# B&R Automation Studio project elevator
Automation Studio 4.2.1.214; Default project

## Configuration Simulation

CPU , AutomationRuntime D4.21

### Hardware
```
PC_any : PC_any v1.1.0.0 (OrderNumber=PC)
  Connector IF3:
    Vnc1
    VncVcObjectName1 = demo
    VncKeyMappingFile1 = VC\PS2-Keyboard.dis
  Cyclic1Duration = 100000
  Cyclic1Tolerance = 10000000
  Cyclic2Duration = 200000
  Cyclic2Tolerance = 10000000
  Cyclic3Duration = 500000
  Cyclic3Tolerance = 10000000
  Cyclic4Duration = 1000000
  Cyclic4Tolerance = 10000000
  Cyclic5Duration = 2000000
  Cyclic5Tolerance = 10000000
  Cyclic6Duration = 3000000
  Cyclic6Tolerance = 12000000
  Cyclic7Duration = 4000000
  Cyclic7Tolerance = 12000000
  Cyclic8Duration = 5000000
  Cyclic8Tolerance = 30000000
```

## Logical view

Binary libraries used (declarations not repeated): Runtime, Operator, AsIecCon, astime, standard, sys_lib, brsystem

### Global.typ - Global data types
```iecst
(*********************************************************************************
 * Copyright:
 * Author:    Chen
 * Created:   April 23, 2016/7:59 PM
 *********************************************************************************
 * Declaration of global data types
 *********************************************************************************)

TYPE

 (*电梯井接口信号定义*)
tTower_Interface: STRUCT

		Sensor_DoorOpened : BOOL;(*传感器信号指示轿厢门已打开*)
		Sensor_DoorClosed : BOOL;(*传感器信号指示轿厢门已关闭*)

		Sensor_Floor1Approached :  BOOL;(*传感器信号指示轿厢已到达对应楼层*)
		Sensor_Floor2Approached :  BOOL;
		Sensor_Floor3Approached :  BOOL;
		Sensor_Floor4Approached :  BOOL;
		Sensor_Floor5Approached :  BOOL;
		Sensor_Floor6Approached :  BOOL;
		Sensor_Floor7Approached :  BOOL;

		Signal_Start_DoorMotor_P : BOOL; (*控制信号，上升沿触发，使轿厢门电机正转固定的角度，打开轿厢门*)
		Signal_Start_DoorMotor_N : BOOL; (*控制信号，上升沿触发，使轿厢门电机反转固定的角度，关闭轿厢门*)

		Signal_Start_CabinMotor_P : BOOL; (*控制信号，上升沿触发，使轿厢提升电机正转，电梯上行*)
		Signal_Start_CabinMotor_N : BOOL; (*控制信号，上升沿触发，使轿厢提升电机反转，电梯下行*)
		Signal_Stop_CabinMotor : BOOL;    (*控制信号，上升沿触发，使轿厢提升电机停止*)

		Sensor_Position_Door : UINT;	  (*轿厢门位置反馈*)
		Sensor_Position_Cabin : UINT;     (*轿厢垂直位置反馈*)

END_STRUCT;

(*楼层面板接口信号定义*)
tFloor_Interface: STRUCT
		Key_Up : BOOL;(*向上按钮*)
		Key_Down : BOOL;(*向下按钮*)
		Display_Current_Floor_Left : USINT;(*左电梯当前楼层显示数码管*)
		Display_Current_Floor_Right : USINT;(*右电梯当前楼层显示数码管*)
		Display_Current_Direction_Left : STRING[2];(*左电梯当前运行方向显示数码管*)
		Display_Current_Direction_Right : STRING[2];(*右电梯当前运行方向显示数码管*)
		Display_UpSelected : tCheckStatus; (*电梯向上按钮指示灯*)
		Display_DownSelected : tCheckStatus; (*电梯向下按钮指示灯*)
END_STRUCT;

(*对应楼层的设置状态*)
tCheckStatus :
		(
		Checked:=16#3340,
		UnChecked:=16#FE10
);

(*轿厢接口信号定义*)
tCabin_Interface: STRUCT

		Key_Open : BOOL; (*开门按钮*)
		Key_Close : BOOL; (*关门按钮*)
		Key_Floor1 : BOOL; (*目标楼层按钮*)
		Key_Floor2 : BOOL;
		Key_Floor3 : BOOL;
		Key_Floor4 : BOOL;
		Key_Floor5 : BOOL;
		Key_Floor6 : BOOL;
		Key_Floor7 : BOOL;
		Display_Floor1Selected : tCheckStatus;(*目标楼层被选中指示灯*)
		Display_Floor2Selected : tCheckStatus;
		Display_Floor3Selected : tCheckStatus;
		Display_Floor4Selected : tCheckStatus;
		Display_Floor5Selected : tCheckStatus;
		Display_Floor6Selected : tCheckStatus;
		Display_Floor7Selected : tCheckStatus;

		Display_Current_Floor : USINT;  (*当前楼层显示数码管*)
		Display_Current_Direction : STRING[2];    (*当前运行方向显示数码管*)

END_STRUCT;

END_TYPE
```

### Global.var - Global variables
```iecst
(*********************************************************************************
 * Copyright:
 * Author:    Chen
 * Created:   April 23, 2016/7:59 PM
 *********************************************************************************
 * Declaration of global variables
 *********************************************************************************)
VAR
	LeftTower : tTower_Interface; (*实例化左电梯井接口*)
	RightTower : tTower_Interface; (*实例化右电梯井接口*)
	LeftCabin : tCabin_Interface; (*实例化左电梯轿厢接口*)
	RightCabin : tCabin_Interface; (*实例化右电梯轿厢接口*)
	FloorPanel : ARRAY[0..6] OF tFloor_Interface := [7(0)];
END_VAR
```


### Program Logical/Model (IEC)

#### Cyclic.st - Cyclic code
```iecst
PROGRAM _CYCLIC

	(*左电梯轿厢门状态机*)
	CASE LeftDoorState OF
		DoorIsClosed:
			IF LeftTower.Signal_Start_DoorMotor_P   THEN
				LeftTower.Sensor_DoorClosed := FALSE;
				LeftDoorState := DoorIsOpening;

			END_IF
		DoorIsOpened:
			IF LeftTower.Signal_Start_DoorMotor_N   THEN
				LeftTower.Sensor_DoorOpened := FALSE;
				LeftDoorState := DoorIsClosing;
			END_IF
		DoorIsClosing:
			IF LeftTower.Sensor_Position_Door > 0 THEN
				LeftTower.Sensor_Position_Door := LeftTower.Sensor_Position_Door-1;
			ELSE
				LeftTower.Sensor_DoorClosed := TRUE;
				LeftDoorState := DoorIsClosed;
			END_IF
		DoorIsOpening:
			IF LeftTower.Sensor_Position_Door < 50 THEN
				LeftTower.Sensor_Position_Door := LeftTower.Sensor_Position_Door+1;
			ELSE
				LeftTower.Sensor_DoorOpened := TRUE;
				LeftDoorState := DoorIsOpened;
			END_IF
	END_CASE

	(*左电梯轿厢运动状态机*)

	CASE LeftCabinState OF
		CabinIsStoped:
			IF LeftTower.Signal_Start_CabinMotor_P   THEN
				LeftCabinState := CabinIsGoingUp;
			ELSIF LeftTower.Signal_Start_CabinMotor_N THEN
				LeftCabinState := CabinIsGoingDown;
			END_IF
			LeftCabin.Display_Current_Direction := '--';
			FOR i := 0 TO 6 DO
				FloorPanel[i].Display_Current_Direction_Left := '--';
			END_FOR
		CabinIsGoingUp:
			IF LeftTower.Sensor_Position_Cabin < 600 THEN
			    LeftTower.Sensor_Position_Cabin := LeftTower.Sensor_Position_Cabin+1;
			END_IF
			IF  LeftTower.Signal_Stop_CabinMotor   THEN
				LeftCabinState := CabinIsStoped;
			END_IF
			LeftCabin.Display_Current_Direction := '/\';
			FOR i := 0 TO 6 DO
				FloorPanel[i].Display_Current_Direction_Left := '/\';
			END_FOR

		CabinIsGoingDown:
			IF LeftTower.Sensor_Position_Cabin > 0 THEN
				LeftTower.Sensor_Position_Cabin := LeftTower.Sensor_Position_Cabin-1;
			END_IF
			IF  LeftTower.Signal_Stop_CabinMotor   THEN
				LeftCabinState := CabinIsStoped;
			END_IF
			LeftCabin.Display_Current_Direction := '\/';
			FOR i := 0 TO 6 DO
				FloorPanel[i].Display_Current_Direction_Left := '\/';
			END_FOR

		END_CASE

	IF LeftTower.Sensor_Position_Cabin = 0 THEN
		LeftTower.Sensor_Floor1Approached := TRUE;
	ELSE
		LeftTower.Sensor_Floor1Approached := FALSE;
	END_IF

	IF LeftTower.Sensor_Position_Cabin = 100 THEN
		LeftTower.Sensor_Floor2Approached := TRUE;
	ELSE
		LeftTower.Sensor_Floor2Approached := FALSE;
	END_IF

	IF LeftTower.Sensor_Position_Cabin = 200 THEN
		LeftTower.Sensor_Floor3Approached := TRUE;
	ELSE
		LeftTower.Sensor_Floor3Approached := FALSE;
	END_IF

	IF LeftTower.Sensor_Position_Cabin = 300 THEN
		LeftTower.Sensor_Floor4Approached := TRUE;
	ELSE
		LeftTower.Sensor_Floor4Approached := FALSE;
	END_IF
	IF LeftTower.Sensor_Position_Cabin = 400 THEN
		LeftTower.Sensor_Floor5Approached := TRUE;
	ELSE
		LeftTower.Sensor_Floor5Approached := FALSE;
	END_IF
	IF LeftTower.Sensor_Position_Cabin = 500 THEN
		LeftTower.Sensor_Floor6Approached := TRUE;
	ELSE
		LeftTower.Sensor_Floor6Approached := FALSE;
	END_IF
	IF LeftTower.Sensor_Position_Cabin = 600 THEN
		LeftTower.Sensor_Floor7Approached := TRUE;
	ELSE
		LeftTower.Sensor_Floor7Approached := FALSE;
	END_IF

	IF LeftTower.Sensor_Position_Cabin < 100 THEN
		LeftCabin.Display_Current_Floor := 1;
	ELSIF 	LeftTower.Sensor_Position_Cabin < 200 THEN
        LeftCabin.Display_Current_Floor := 2;
	ELSIF 	LeftTower.Sensor_Position_Cabin < 300 THEN
		LeftCabin.Display_Current_Floor := 3;
	ELSIF 	LeftTower.Sensor_Position_Cabin < 400 THEN
		LeftCabin.Display_Current_Floor := 4;
	ELSIF 	LeftTower.Sensor_Position_Cabin < 500 THEN
		LeftCabin.Display_Current_Floor := 5;
	ELSIF 	LeftTower.Sensor_Position_Cabin < 600 THEN
		LeftCabin.Display_Current_Floor := 6;
	ELSE
		LeftCabin.Display_Current_Floor := 7;
	END_IF

	FOR i := 0 TO 6 DO
		FloorPanel[i].Display_Current_Floor_Left := LeftCabin.Display_Current_Floor;
	END_FOR

	(*右电梯轿厢门状态机*)
	CASE RightDoorState OF
		DoorIsClosed:
			IF RightTower.Signal_Start_DoorMotor_P   THEN
				RightTower.Sensor_DoorClosed := FALSE;
				RightDoorState := DoorIsOpening;

			END_IF
		DoorIsOpened:
			IF RightTower.Signal_Start_DoorMotor_N   THEN
				RightTower.Sensor_DoorOpened := FALSE;
				RightDoorState := DoorIsClosing;
			END_IF
		DoorIsClosing:
			IF RightTower.Sensor_Position_Door > 0 THEN
				RightTower.Sensor_Position_Door := RightTower.Sensor_Position_Door-1;
			ELSE
				RightTower.Sensor_DoorClosed := TRUE;
				RightDoorState := DoorIsClosed;
			END_IF
		DoorIsOpening:
			IF RightTower.Sensor_Position_Door < 50 THEN
				RightTower.Sensor_Position_Door := RightTower.Sensor_Position_Door+1;
			ELSE
				RightTower.Sensor_DoorOpened := TRUE;
				RightDoorState := DoorIsOpened;
			END_IF
	END_CASE

	(*右电梯轿厢运动状态机*)

	CASE RightCabinState OF
		CabinIsStoped:
			IF RightTower.Signal_Start_CabinMotor_P   THEN
				RightCabinState := CabinIsGoingUp;
			ELSIF RightTower.Signal_Start_CabinMotor_N THEN
				RightCabinState := CabinIsGoingDown;
			END_IF
			RightCabin.Display_Current_Direction := '--';
			FOR i := 0 TO 6 DO
				FloorPanel[i].Display_Current_Direction_Right := '--';
			END_FOR

		CabinIsGoingUp:
			IF RightTower.Sensor_Position_Cabin < 600 THEN
				RightTower.Sensor_Position_Cabin := RightTower.Sensor_Position_Cabin+1;
			END_IF
			IF  RightTower.Signal_Stop_CabinMotor   THEN
				RightCabinState := CabinIsStoped;
			END_IF
			RightCabin.Display_Current_Direction := '/\';
			FOR i := 0 TO 6 DO
				FloorPanel[i].Display_Current_Direction_Right := '/\';
			END_FOR

		CabinIsGoingDown:
			IF RightTower.Sensor_Position_Cabin > 0 THEN
				RightTower.Sensor_Position_Cabin := RightTower.Sensor_Position_Cabin-1;
			END_IF
			IF  RightTower.Signal_Stop_CabinMotor   THEN
				RightCabinState := CabinIsStoped;
			END_IF
			RightCabin.Display_Current_Direction := '\/';
			FOR i := 0 TO 6 DO
				FloorPanel[i].Display_Current_Direction_Right := '\/';
			END_FOR

	END_CASE

	IF RightTower.Sensor_Position_Cabin = 0 THEN
		RightTower.Sensor_Floor1Approached := TRUE;
	ELSE
		RightTower.Sensor_Floor1Approached := FALSE;
	END_IF

	IF RightTower.Sensor_Position_Cabin = 100 THEN
		RightTower.Sensor_Floor2Approached := TRUE;
	ELSE
		RightTower.Sensor_Floor2Approached := FALSE;
	END_IF

	IF RightTower.Sensor_Position_Cabin = 200 THEN
		RightTower.Sensor_Floor3Approached := TRUE;
	ELSE
		RightTower.Sensor_Floor3Approached := FALSE;
	END_IF

	IF RightTower.Sensor_Position_Cabin = 300 THEN
		RightTower.Sensor_Floor4Approached := TRUE;
	ELSE
		RightTower.Sensor_Floor4Approached := FALSE;
	END_IF
	IF RightTower.Sensor_Position_Cabin = 400 THEN
		RightTower.Sensor_Floor5Approached := TRUE;
	ELSE
		RightTower.Sensor_Floor5Approached := FALSE;
	END_IF
	IF RightTower.Sensor_Position_Cabin = 500 THEN
		RightTower.Sensor_Floor6Approached := TRUE;
	ELSE
		RightTower.Sensor_Floor6Approached := FALSE;
	END_IF
	IF RightTower.Sensor_Position_Cabin = 600 THEN
		RightTower.Sensor_Floor7Approached := TRUE;
	ELSE
		RightTower.Sensor_Floor7Approached := FALSE;
	END_IF

	IF RightTower.Sensor_Position_Cabin < 100 THEN
		RightCabin.Display_Current_Floor := 1;
	ELSIF 	RightTower.Sensor_Position_Cabin < 200 THEN
		RightCabin.Display_Current_Floor := 2;
	ELSIF 	RightTower.Sensor_Position_Cabin < 300 THEN
		RightCabin.Display_Current_Floor := 3;
	ELSIF 	RightTower.Sensor_Position_Cabin < 400 THEN
		RightCabin.Display_Current_Floor := 4;
	ELSIF 	RightTower.Sensor_Position_Cabin < 500 THEN
		RightCabin.Display_Current_Floor := 5;
	ELSIF 	RightTower.Sensor_Position_Cabin < 600 THEN
		RightCabin.Display_Current_Floor := 6;
	ELSE
		RightCabin.Display_Current_Floor := 7;
	END_IF
	FOR i := 0 TO 6 DO
		FloorPanel[i].Display_Current_Floor_Right := RightCabin.Display_Current_Floor;
	END_FOR

END_PROGRAM
```

#### Init.st - Init code
```iecst
PROGRAM _INIT
	(* Insert code here *)
	LeftDoorState := DoorIsClosed;
	LeftCabinState := CabinIsStoped;

	LeftTower.Sensor_DoorClosed := TRUE;
	LeftTower.Sensor_DoorOpened := FALSE;
	LeftTower.Sensor_Floor1Approached := TRUE;
	LeftTower.Sensor_Floor2Approached := FALSE;
	LeftTower.Sensor_Floor3Approached := FALSE;
	LeftTower.Sensor_Floor4Approached := FALSE;
	LeftTower.Sensor_Floor5Approached := FALSE;
	LeftTower.Sensor_Floor6Approached := FALSE;
	LeftTower.Sensor_Floor7Approached := FALSE;
	LeftTower.Sensor_Position_Door := 0;
	LeftTower.Sensor_Position_Cabin := 0;

	LeftCabin.Display_Current_Direction := '--';
	RightCabin.Display_Current_Direction := '--';

END_PROGRAM
```

#### Types.typ - Local data types
```iecst
TYPE
tDoorState :
(
	DoorIsClosed,
	DoorIsOpened,
	DoorIsClosing,
	DoorIsOpening
);

tCabinState :
(
	CabinIsStoped,
	CabinIsGoingUp,
	CabinIsGoingDown
);
END_TYPE
```

#### Variables.var - Local variables
```iecst
VAR
	Current_Direction_Left : USINT := 1;
	Current_Direction_Right : USINT := 1;
	Current_Floor_Left : USINT := 1;
	Current_Floor_Right : USINT := 1;
	disp_direction : STRING[2] := '';
	i : USINT := 0;
	Key_Close_Left : BOOL := FALSE;
	Key_Close_Right : BOOL := FALSE;
	Key_Down_Floor1 : BOOL := FALSE;
	Key_Down_Floor2 : BOOL := FALSE;
	Key_Down_Floor3 : BOOL := FALSE;
	Key_Down_Floor4 : BOOL := FALSE;
	Key_Down_Floor5 : BOOL := FALSE;
	Key_Down_Floor6 : BOOL := FALSE;
	Key_Down_Floor7 : BOOL := FALSE;
	Key_Floor1_Left : BOOL := FALSE;
	Key_Floor1_Right : BOOL := FALSE;
	Key_Floor2_Left : BOOL := FALSE;
	Key_Floor2_Right : BOOL := FALSE;
	Key_Floor3_Left : BOOL := FALSE;
	Key_Floor3_Right : BOOL := FALSE;
	Key_Floor4_Left : BOOL := FALSE;
	Key_Floor4_Right : BOOL := FALSE;
	Key_Floor5_Left : BOOL := FALSE;
	Key_Floor5_Right : BOOL := FALSE;
	Key_Floor6_Left : BOOL := FALSE;
	Key_Floor6_Right : BOOL := FALSE;
	Key_Floor7_Left : BOOL := FALSE;
	Key_Floor7_Right : BOOL := FALSE;
	Key_Open_Left : BOOL := FALSE;
	Key_Open_Right : BOOL := FALSE;
	Key_Up_Floor1 : BOOL := FALSE;
	Key_Up_Floor2 : BOOL := FALSE;
	Key_Up_Floor3 : BOOL := FALSE;
	Key_Up_Floor4 : BOOL := FALSE;
	Key_Up_Floor5 : BOOL := FALSE;
	Key_Up_Floor6 : BOOL := FALSE;
	Key_Up_Floor7 : BOOL := FALSE;
	LeftCabinState : tCabinState;
	LeftDoorState : tDoorState;
	Position_Cabin_Left : UINT := 0;
	Position_Cabin_Right : UINT := 0;
	Position_Door_Left : UINT := 0;
	Position_Door_Right : UINT := 0;
	RightCabinState : tCabinState;
	RightDoorState : tDoorState;
	Sensor_Closed_Left : BOOL := FALSE;
	Sensor_Closed_Right : BOOL := FALSE;
	Sensor_Floor1_Left : BOOL := FALSE;
	Sensor_Floor1_Right : BOOL := FALSE;
	Sensor_Floor2_Left : BOOL := FALSE;
	Sensor_Floor2_Right : BOOL := FALSE;
	Sensor_Floor3_Left : BOOL := FALSE;
	Sensor_Floor3_Right : BOOL := FALSE;
	Sensor_Floor4_Left : BOOL := FALSE;
	Sensor_Floor4_Right : BOOL := FALSE;
	Sensor_Floor5_Left : BOOL := FALSE;
	Sensor_Floor5_Right : BOOL := FALSE;
	Sensor_Floor6_Left : BOOL := FALSE;
	Sensor_Floor6_Right : BOOL := FALSE;
	Sensor_Floor7_Left : BOOL := FALSE;
	Sensor_Floor7_Right : BOOL := FALSE;
	Sensor_Opened_Left : BOOL := FALSE;
	Sensor_Opened_Right : BOOL := FALSE;
	Target_Floor_Left : USINT := 1;
	Target_Floor_Right : USINT := 1;
END_VAR
```

- Visualisation Logical/demo (not shown)

### Program Logical/controller (IEC)

#### Variables.var
```iecst
VAR
	DownLast : USINT := 0;
	UpLast : USINT := 0;
	i : USINT := 0;
	j : USINT := 0;
	k : USINT := 0;
	UpList : ARRAY[0..6] OF USINT := [7(0)];
	DownList : ARRAY[0..6] OF USINT := [7(0)];
END_VAR
```

#### Cyclic.st
```iecst
PROGRAM _CYCLIC
	(* Insert code here *)
	(*下列代码只是为了测试*)

	LeftTower.Signal_Start_DoorMotor_P := LeftCabin.Key_Open ;
	LeftTower.Signal_Start_DoorMotor_N := LeftCabin.Key_Close ;

	RightTower.Signal_Start_DoorMotor_P := RightCabin.Key_Open ;
	RightTower.Signal_Start_DoorMotor_N := RightCabin.Key_Close ;

//refresh the UpList
	FOR i := 0 TO 6 DO
		IF UpList[i] = 0 THEN
			UpLast := i;
			EXIT;
		END_IF
	END_FOR

	FOR i := 0 TO 6 DO
		IF FloorPanel[i].Key_Up THEN
			FOR j := 0 TO 6 DO
				IF UpList[j] = i+1 THEN
					EXIT;
				END_IF
				IF j = 6 THEN
					UpList[UpLast] := i+1;
					UpLast := UpLast+1;
				END_IF
			END_FOR
		END_IF
	END_FOR
//refresh the DownList
	FOR i := 0 TO 6 DO
		IF DownList[i] = 0 THEN
			DownLast := i;
			EXIT;
		END_IF
	END_FOR

	FOR i := 0 TO 6 DO
		IF FloorPanel[i].Key_Down THEN
			FOR j := 0 TO 6 DO
				IF DownList[j] = i+1 THEN
					EXIT;
				END_IF
				IF j = 6 THEN
					DownList[DownLast] := i+1;
					DownLast := DownLast+1;
				END_IF
			END_FOR
		END_IF
	END_FOR
	IF UpList[0] <> 0 THEN
		IF LeftCabin.Display_Current_Floor < UpList[0] THEN
			LeftTower.Signal_Start_CabinMotor_P := TRUE;
			LeftTower.Signal_Start_CabinMotor_N := FALSE;
		END_IF
		IF LeftCabin.Display_Current_Floor > UpList[0] THEN
			LeftTower.Signal_Start_CabinMotor_N := TRUE;
			LeftTower.Signal_Start_CabinMotor_N := FALSE;
		END_IF
		IF LeftCabin.Display_Current_Floor = UpList[0] THEN
			LeftTower.Signal_Stop_CabinMotor := TRUE;
			LeftTower.Signal_Start_CabinMotor_P := FALSE;
			LeftTower.Signal_Start_CabinMotor_N := FALSE;
			LeftTower.Signal_Start_DoorMotor_P := TRUE;
			FOR i := 0 TO 6 DO
				UpList[i] := UpList[i+1] ;
				EXIT;
				END_FOR
		END_IF
	END_IF

//	LeftTower.Signal_Start_CabinMotor_P := FloorPanel[0].Key_Up ;
//	RightTower.Signal_Start_CabinMotor_P := FloorPanel[0].Key_Up ;
//
//	LeftTower.Signal_Start_CabinMotor_N := FloorPanel[6].Key_Down ;
//	RightTower.Signal_Start_CabinMotor_N := FloorPanel[6].Key_Down ;
//
//	LeftTower.Signal_Stop_CabinMotor := FloorPanel[3].Key_Up ;
//	RightTower.Signal_Stop_CabinMotor := FloorPanel[3].Key_Up ;

	IF LeftCabin.Display_Floor1Selected = UnChecked AND LeftCabin.Key_Floor1 =1 THEN
		LeftCabin.Display_Floor1Selected := Checked;
	END_IF
	IF LeftCabin.Display_Floor2Selected = UnChecked AND LeftCabin.Key_Floor2 =1 THEN
		LeftCabin.Display_Floor2Selected := Checked;
	END_IF
	IF LeftCabin.Display_Floor3Selected = UnChecked AND LeftCabin.Key_Floor3 =1 THEN
		LeftCabin.Display_Floor3Selected := Checked;
	END_IF
	IF LeftCabin.Display_Floor4Selected = UnChecked AND LeftCabin.Key_Floor4 =1 THEN
		LeftCabin.Display_Floor4Selected := Checked;
	END_IF
	IF LeftCabin.Display_Floor5Selected = UnChecked AND LeftCabin.Key_Floor5 =1 THEN
		LeftCabin.Display_Floor5Selected := Checked;
	END_IF
	IF LeftCabin.Display_Floor6Selected = UnChecked AND LeftCabin.Key_Floor6 =1 THEN
		LeftCabin.Display_Floor6Selected := Checked;
	END_IF
	IF LeftCabin.Display_Floor7Selected = UnChecked AND LeftCabin.Key_Floor7 =1 THEN
		LeftCabin.Display_Floor7Selected := Checked;
	END_IF

	IF RightCabin.Display_Floor1Selected = UnChecked AND RightCabin.Key_Floor1 =1 THEN
		RightCabin.Display_Floor1Selected := Checked;
	END_IF
	IF RightCabin.Display_Floor2Selected = UnChecked AND RightCabin.Key_Floor2 =1 THEN
		RightCabin.Display_Floor2Selected := Checked;
	END_IF
	IF RightCabin.Display_Floor3Selected = UnChecked AND RightCabin.Key_Floor3 =1 THEN
		RightCabin.Display_Floor3Selected := Checked;
	END_IF
	IF RightCabin.Display_Floor4Selected = UnChecked AND RightCabin.Key_Floor4 =1 THEN
		RightCabin.Display_Floor4Selected := Checked;
	END_IF
	IF RightCabin.Display_Floor5Selected = UnChecked AND RightCabin.Key_Floor5 =1 THEN
		RightCabin.Display_Floor5Selected := Checked;
	END_IF
	IF RightCabin.Display_Floor6Selected = UnChecked AND RightCabin.Key_Floor6 =1 THEN
		RightCabin.Display_Floor6Selected := Checked;
	END_IF
	IF RightCabin.Display_Floor7Selected = UnChecked AND RightCabin.Key_Floor7 =1 THEN
		RightCabin.Display_Floor7Selected := Checked;
	END_IF

END_PROGRAM
```

#### Cyclic1.ld
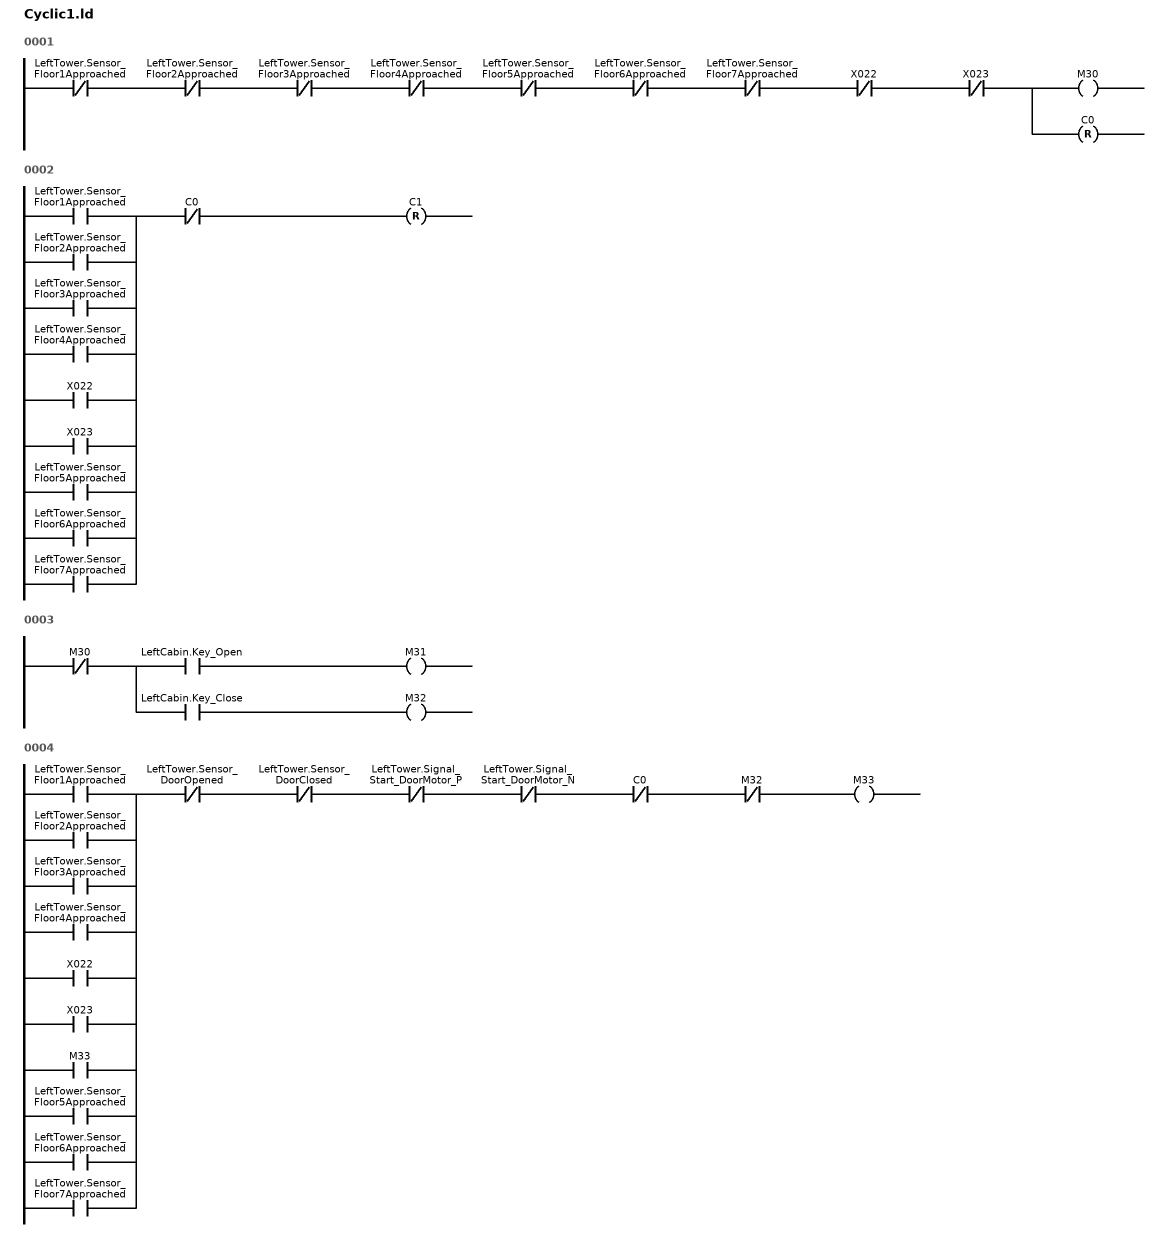
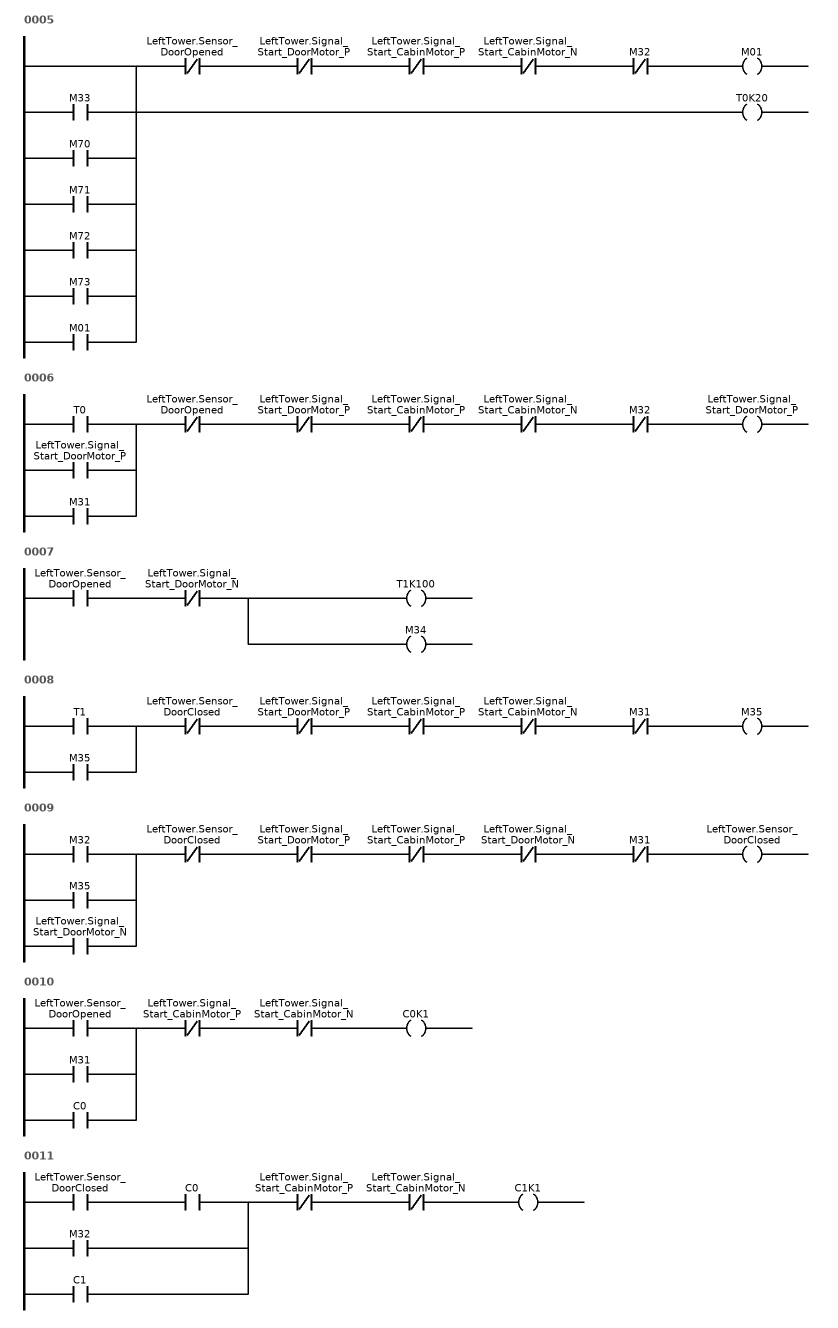
Ladder, written as Structured Text:
```iecst
PROGRAM _CYCLIC
VAR
    _p1 : BOOL;
    _z2 : BOOL;
    _z3 : BOOL;
    _z4 : BOOL;
    _z5 : BOOL;
    _z6 : BOOL;
    _z7 : BOOL;
    _p8 : BOOL;
    _p9 : BOOL;
END_VAR
(* Network 1 *)
_p1 := NOT LeftTower.Sensor_Floor1Approached AND NOT LeftTower.Sensor_Floor2Approached AND NOT LeftTower.Sensor_Floor3Approached AND NOT LeftTower.Sensor_Floor4Approached AND NOT LeftTower.Sensor_Floor5Approached AND NOT LeftTower.Sensor_Floor6Approached AND NOT LeftTower.Sensor_Floor7Approached AND NOT X022 AND NOT X023;
M30 := _p1;
IF _p1 THEN C0 := FALSE; END_IF;

(* Network 2 *)
IF (LeftTower.Sensor_Floor1Approached OR LeftTower.Sensor_Floor2Approached OR LeftTower.Sensor_Floor3Approached OR LeftTower.Sensor_Floor4Approached OR X022 OR X023 OR LeftTower.Sensor_Floor5Approached OR LeftTower.Sensor_Floor6Approached OR LeftTower.Sensor_Floor7Approached) AND NOT C0 THEN
    C1 := FALSE;
END_IF;

(* Network 3 *)
M31 := NOT M30 AND LeftCabin.Key_Open;
M32 := NOT M30 AND LeftCabin.Key_Close;

(* Network 4 *)
M33 := (LeftTower.Sensor_Floor1Approached OR LeftTower.Sensor_Floor2Approached OR LeftTower.Sensor_Floor3Approached OR LeftTower.Sensor_Floor4Approached OR X022 OR X023 OR M33 OR LeftTower.Sensor_Floor5Approached OR LeftTower.Sensor_Floor6Approached OR LeftTower.Sensor_Floor7Approached) AND NOT LeftTower.Sensor_DoorOpened AND NOT LeftTower.Sensor_DoorClosed AND NOT LeftTower.Signal_Start_DoorMotor_P AND NOT LeftTower.Signal_Start_DoorMotor_N AND NOT C0 AND NOT M32;

(* Network 5 *)
_z7 := M01;
_z6 := M73;
_z5 := M72;
_z4 := M71;
_z3 := M70;
_z2 := M33;
_p8 := M01;
M01 := NOT LeftTower.Sensor_DoorOpened AND NOT LeftTower.Signal_Start_DoorMotor_P AND NOT LeftTower.Signal_Start_CabinMotor_P AND NOT LeftTower.Signal_Start_CabinMotor_N AND NOT M32;
T0K20 := TRUE;

(* Network 6 *)
LeftTower.Signal_Start_DoorMotor_P := (T0 OR LeftTower.Signal_Start_DoorMotor_P OR M31) AND NOT LeftTower.Sensor_DoorOpened AND NOT LeftTower.Signal_Start_DoorMotor_P AND NOT LeftTower.Signal_Start_CabinMotor_P AND NOT LeftTower.Signal_Start_CabinMotor_N AND NOT M32;

(* Network 7 *)
_p9 := LeftTower.Sensor_DoorOpened AND NOT LeftTower.Signal_Start_DoorMotor_N;
T1K100 := _p9;
M34 := _p9;

(* Network 8 *)
M35 := (T1 OR M35) AND NOT LeftTower.Sensor_DoorClosed AND NOT LeftTower.Signal_Start_DoorMotor_P AND NOT LeftTower.Signal_Start_CabinMotor_P AND NOT LeftTower.Signal_Start_CabinMotor_N AND NOT M31;

(* Network 9 *)
LeftTower.Sensor_DoorClosed := (M32 OR M35 OR LeftTower.Signal_Start_DoorMotor_N) AND NOT LeftTower.Sensor_DoorClosed AND NOT LeftTower.Signal_Start_DoorMotor_P AND NOT LeftTower.Signal_Start_CabinMotor_P AND NOT LeftTower.Signal_Start_DoorMotor_N AND NOT M31;

(* Network 10 *)
C0K1 := (LeftTower.Sensor_DoorOpened OR M31 OR C0) AND NOT LeftTower.Signal_Start_CabinMotor_P AND NOT LeftTower.Signal_Start_CabinMotor_N;

(* Network 11 *)
C1K1 := ((LeftTower.Sensor_DoorClosed AND C0) OR M32 OR C1) AND NOT LeftTower.Signal_Start_CabinMotor_P AND NOT LeftTower.Signal_Start_CabinMotor_N;
END_PROGRAM
```

#### Init.st
```iecst
PROGRAM _INIT
	(* Insert code here *)
	LeftCabin.Display_Floor1Selected := UnChecked;
	LeftCabin.Display_Floor2Selected := UnChecked;
	LeftCabin.Display_Floor3Selected := UnChecked;
	LeftCabin.Display_Floor4Selected := UnChecked;
	LeftCabin.Display_Floor5Selected := UnChecked;
	LeftCabin.Display_Floor6Selected := UnChecked;
	LeftCabin.Display_Floor7Selected := UnChecked;

	RightCabin.Display_Floor1Selected := UnChecked;
	RightCabin.Display_Floor2Selected := UnChecked;
	RightCabin.Display_Floor3Selected := UnChecked;
	RightCabin.Display_Floor4Selected := UnChecked;
	RightCabin.Display_Floor5Selected := UnChecked;
	RightCabin.Display_Floor6Selected := UnChecked;
	RightCabin.Display_Floor7Selected := UnChecked;

END_PROGRAM
```

Listed in the project but not available here: Logical/Model/Exit.st
